# EPICS IOC start-up script: iocsh/ethercatmcAuxBitAsMbbiRecord.iocsh
dbLoadRecords("ethercatmcAuxBitAsMbbiRecord.template", "PREFIX=$(PREFIX), MOTOR_NAME=$(MOTOR_NAME), MOTOR_PORT=$(MOTOR_PORT), AXIS_NO=$(AXIS_NO), AUXBITS07=$(AUXBITS07)")
